{attribute 'linkalways'} 
{attribute 'no_explicit_call' := 'This FB is a CLASS and must be accessed using methods or properties'}
{attribute 'enable_dynamic_creation'}
FUNCTION_BLOCK _ETcVnFontType EXTENDS EnumDatatypeBase
VAR
	localData : ETcVnFontType;
	activeData : REFERENCE TO ETcVnFontType;
	enumBaseDatatype : _DINT(localData);
END_VAR

METHOD PRIVATE AddLocalEnumeration
VAR_INPUT
	Enumeration : T_MAXSTRING;
	Value : ETcVnFontType;
END_VAR
AddEnumeration(Enumeration, Value);
END_METHOD

PROPERTY PUBLIC Address : PVOID
GET
Address := ADR(activeData);
END_GET
END_PROPERTY

METHOD PUBLIC ClearReference
VAR_INPUT
END_VAR
activeData REF= localData;
SetBaseDatatypeReference();
END_METHOD

METHOD PUBLIC Clone : I_Datatype
VAR
    pClone : POINTER TO _ETcVnFontType;
END_VAR
pClone := __NEW(_ETcVnFontType(InitialValue := Value));
Clone := pClone^;
END_METHOD

METHOD FB_init : BOOL
VAR_INPUT
	bInitRetains : BOOL; // if TRUE, the retain variables are initialized (warm start / cold start)
	bInCopyCode : BOOL;  // if TRUE, the instance afterwards gets moved into the copy code (online change)
	InitialValue : ETcVnFontType;
END_VAR
localData := InitialValue;
AddBaseDatatype(enumBaseDatatype);
ClearReference();

AddLocalEnumeration('TCVN_FT_HERSHEY_SIMPLEX', ETcVnFontType.TCVN_FT_HERSHEY_SIMPLEX);
AddLocalEnumeration('TCVN_FT_HERSHEY_PLAIN', ETcVnFontType.TCVN_FT_HERSHEY_PLAIN);
AddLocalEnumeration('TCVN_FT_HERSHEY_DUPLEX', ETcVnFontType.TCVN_FT_HERSHEY_DUPLEX);
AddLocalEnumeration('TCVN_FT_HERSHEY_COMPLEX', ETcVnFontType.TCVN_FT_HERSHEY_COMPLEX);
AddLocalEnumeration('TCVN_FT_HERSHEY_TRIPLEX', ETcVnFontType.TCVN_FT_HERSHEY_TRIPLEX);
AddLocalEnumeration('TCVN_FT_HERSHEY_COMPLEX_SMALL', ETcVnFontType.TCVN_FT_HERSHEY_COMPLEX_SMALL);
AddLocalEnumeration('TCVN_FT_HERSHEY_SCRIPT_SIMPLEX', ETcVnFontType.TCVN_FT_HERSHEY_SCRIPT_SIMPLEX);
AddLocalEnumeration('TCVN_FT_HERSHEY_SCRIPT_COMPLEX', ETcVnFontType.TCVN_FT_HERSHEY_SCRIPT_COMPLEX);
AddLocalEnumeration('TCVN_FT_HERSHEY_PLAIN_ITALIC', ETcVnFontType.TCVN_FT_HERSHEY_PLAIN_ITALIC);
AddLocalEnumeration('TCVN_FT_HERSHEY_COMPLEX_ITALIC', ETcVnFontType.TCVN_FT_HERSHEY_COMPLEX_ITALIC);
AddLocalEnumeration('TCVN_FT_HERSHEY_TRIPLEX_ITALIC', ETcVnFontType.TCVN_FT_HERSHEY_TRIPLEX_ITALIC);
AddLocalEnumeration('TCVN_FT_HERSHEY_COMPLEX_SMALL_ITALIC', ETcVnFontType.TCVN_FT_HERSHEY_COMPLEX_SMALL_ITALIC);
END_METHOD

PROPERTY PUBLIC Identifier : T_MAXSTRING
GET
Identifier := 'ETcVnFontType';
END_GET
END_PROPERTY

METHOD IsEnumeratorValueEqual : BOOL
VAR_INPUT
	Enumerator : I_KeyValueForwardEnumerator;
END_VAR
VAR
	storedValue : ETcVnFontType;
END_VAR
IF NOT Enumerator.TryGet(storedValue) THEN
	RETURN;
END_IF

IsEnumeratorValueEqual := storedValue = activeData;
END_METHOD

METHOD PUBLIC MakeReferenceTo
VAR_INPUT
	ReferenceTarget : REFERENCE TO ETcVnFontType;
END_VAR
activeData REF= ReferenceTarget;
SetBaseDatatypeReference();
END_METHOD

METHOD PROTECTED SetBaseDatatypeReference
VAR_INPUT
END_VAR
enumBaseDatatype.MakeReferenceTo(activeData);
END_METHOD

PROPERTY PUBLIC Size : UDINT
GET
Size := SIZEOF(activeData);
END_GET
END_PROPERTY

METHOD TryMakeReferenceTo : BOOL
VAR_INPUT
	Target : I_Datatype;
END_VAR
VAR
	pTargetData : POINTER TO ETcVnFontType;
END_VAR
IF NOT IsEquivalentTo(Target) THEN
	RETURN;
END_IF

pTargetData := Target.Address;
activeData REF= pTargetData^;
SetBaseDatatypeReference();
TryMakeReferenceTo := TRUE;
END_METHOD

PROPERTY PUBLIC Value : ETcVnFontType
GET
Value := activeData;
END_GET
SET
activeData := Value;
END_SET
END_PROPERTY

END_FUNCTION_BLOCK

(* stored: Version 1.1.0.1, ProductVersion 3.1.4024.13
   POU _ETcVnFontType: Id {a73b5c24-6eb0-02a8-1d8c-f6047a4e72cb}, SpecialFunc None
   Folder Core: Id {00d2baa3-5177-08b3-348e-917c2b1004b6}
   Folder Protected: Id {875bedc7-5821-0555-0dd4-7b4f0b34d7c7}
   Folder Customize: Id {4008137c-d89b-0a25-227a-777a536c3165}
   Folder Constructor: Id {740b811e-ba9a-01dc-246b-dbbcd957aedd}
   Folder Private: Id {5fe382ba-e63a-06dd-2af0-09b47c622f91}
   Folder Protected: Id {5d44a6b8-75eb-09de-1d05-22f23d45f459}
   Method AddLocalEnumeration: Id {474cb5f3-f0c6-0d0a-2bb4-80f75f0b16d9}
   Property Address: Id {45d7abf1-877d-08d0-16ad-9dbc38cb74e5}
   Get Get: Id {2b6876a2-fb9b-0409-0a16-2979341491fc}
   Method ClearReference: Id {19804776-82d6-006e-25d7-d241a234ec49}
   Method Clone: Id {e3d5b0da-bc01-0f2f-20fc-9bd718a6c910}
   Method FB_init: Id {f26bf505-a1ca-0583-2055-fe5ba91154bd}
   Property Identifier: Id {8d35aefd-c1c2-03aa-13bf-dc743cc5ac85}
   Get Get: Id {f8dce83b-4a56-069e-3d68-4491395e9524}
   Method IsEnumeratorValueEqual: Id {84dcb567-4289-081f-2dd7-1b8d5a7da990}
   Method MakeReferenceTo: Id {8364ee4f-b8ae-0238-2745-92d173a7ff8e}
   Method SetBaseDatatypeReference: Id {9a2c2350-8ed7-0cc3-0b57-d75b5f831d34}
   Property Size: Id {7ed34594-133d-0457-3d17-280316fa7eac}
   Get Get: Id {2301a4ce-3ac2-098b-2e5d-0a0d8161c4b3}
   Method TryMakeReferenceTo: Id {03e4317d-4353-09ad-05a7-cced2c3a6d17}
   Property Value: Id {ac4e2c3d-0109-043e-354d-8a8bcfaa5827}
   Get Get: Id {093a260e-785c-0240-13bd-3fa61d32b9a9}
   Set Set: Id {7209e334-97db-0abf-1020-e8a50c022862} *)
